SUBAPPLICATION Maehwerksklappung_DM (* Mähwerksklappung Aufgabe Febr. 2026 *)
  (* Standard: 61499-2 *)
  (* Version 1.0, 2026-02-23, Herr Lehrer *)
  PACKAGE Meins;
  IMPORT logiBUS::io::DI::logiBUS_DI::Input_I1;
  IMPORT logiBUS::io::DI::logiBUS_DI::Input_I2;
  IMPORT logiBUS::io::DI::logiBUS_DI::Input_I3;
  IMPORT logiBUS::io::DI::logiBUS_DI::Input_I4;
  IMPORT logiBUS::io::DI::logiBUS_DI::Input_I5;
  IMPORT logiBUS::io::DI::logiBUS_DI::Input_I6;
  IMPORT logiBUS::io::DI::logiBUS_DI_Events::BUTTON_PRESS_DOWN;
  IMPORT logiBUS::io::DI::logiBUS_DI_Events::BUTTON_PRESS_UP;
  IMPORT logiBUS::io::DI::logiBUS_DI_Events::BUTTON_SINGLE_CLICK;
  IMPORT logiBUS::io::DQ::logiBUS_DO::Output_Q1;
  IMPORT logiBUS::io::DQ::logiBUS_DO::Output_Q2;
  IMPORT logiBUS::io::DQ::logiBUS_DO::Output_Q3;
  IMPORT logiBUS::io::DQ::logiBUS_DO::Output_Q4;
  IMPORT logiBUS::io::DQ::logiBUS_DO::Output_Q5;
  IMPORT logiBUS::io::DQ::logiBUS_DO::Output_Q6;
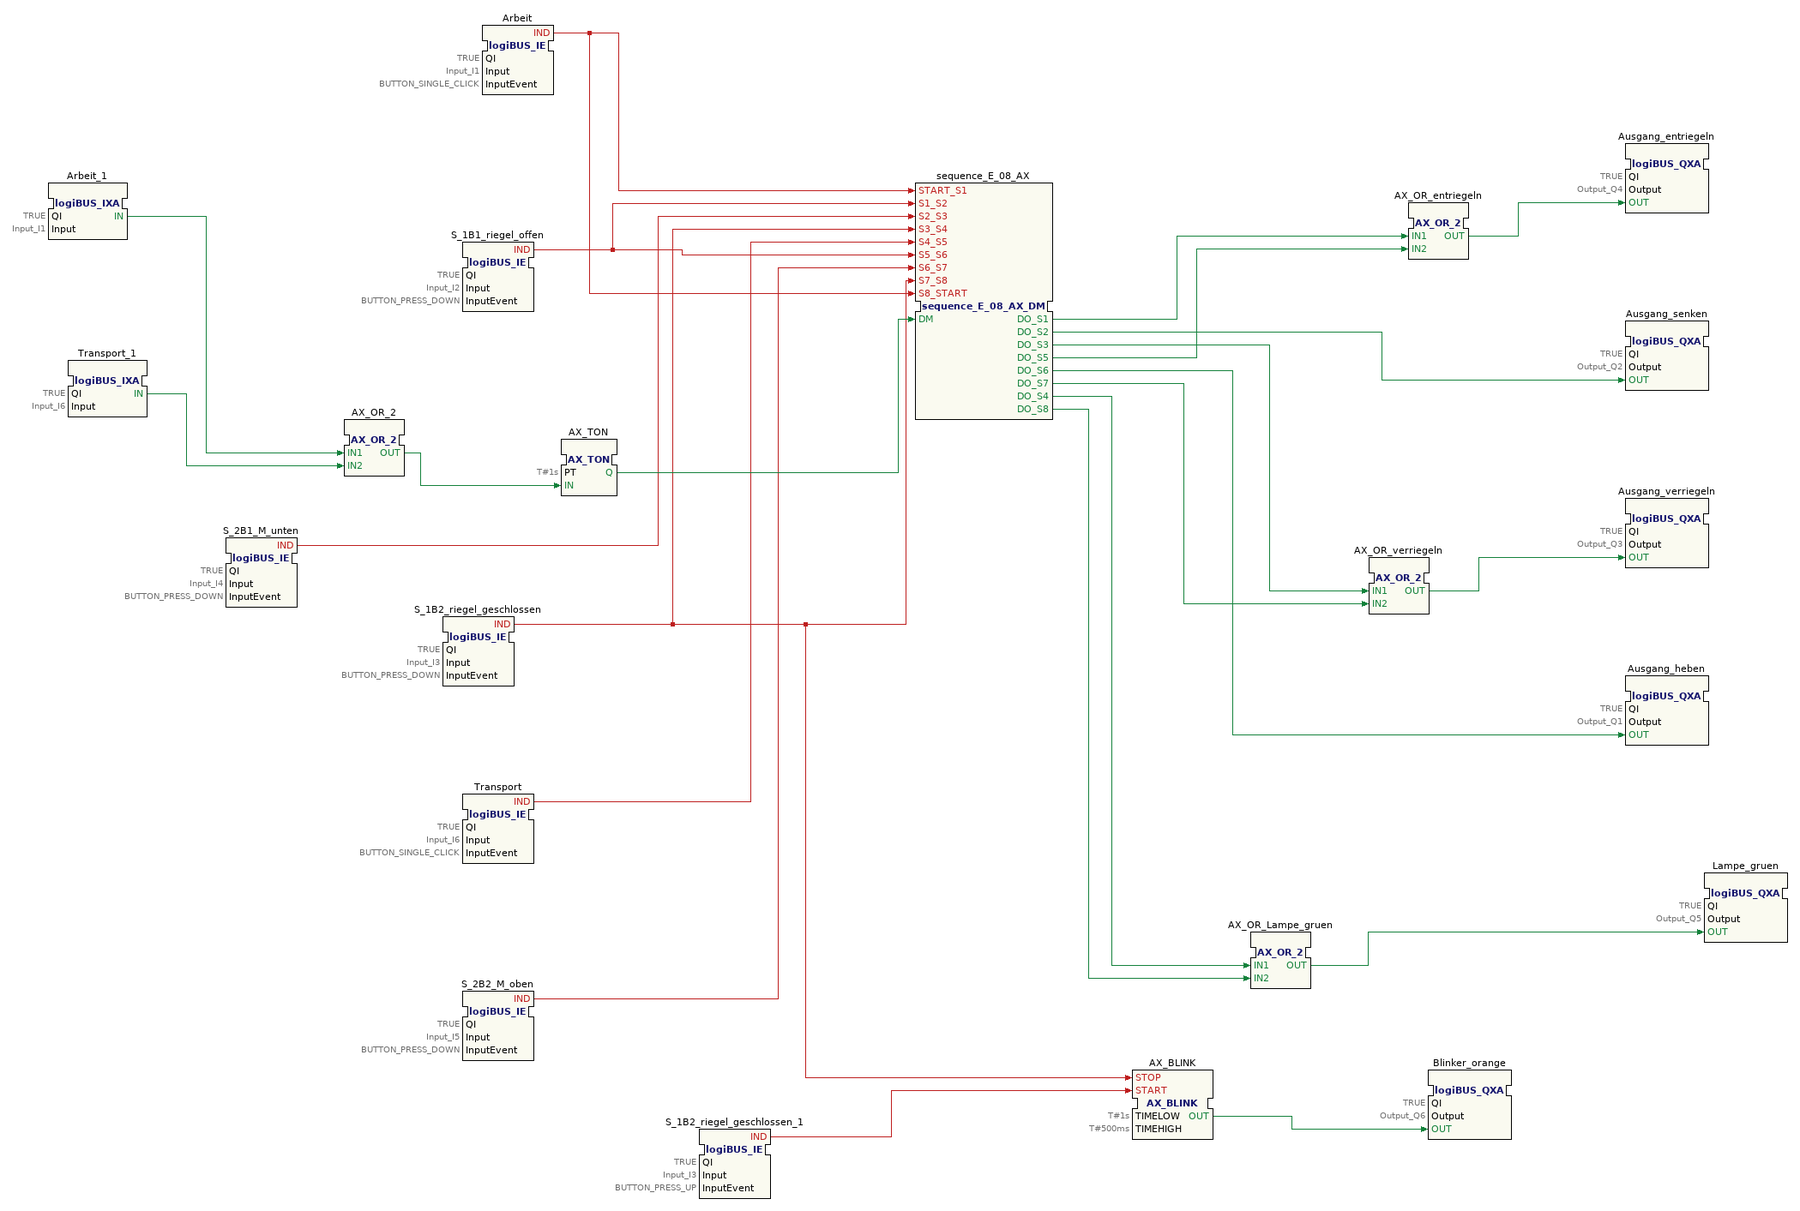
  (* UNTEN *)
  (* S4 ist der Zustand "Arbeit" *)
  (* S8 ist Zustand "Transport" *)
  FBS
    Ausgang_heben : logiBUS::io::DQ::logiBUS_QXA(QI := TRUE, Output := Output_Q1);
    Ausgang_senken : logiBUS::io::DQ::logiBUS_QXA(QI := TRUE, Output := Output_Q2);
    Ausgang_entriegeln : logiBUS::io::DQ::logiBUS_QXA(QI := TRUE, Output := Output_Q4);
    Ausgang_verriegeln : logiBUS::io::DQ::logiBUS_QXA(QI := TRUE, Output := Output_Q3);
    Lampe_gruen : logiBUS::io::DQ::logiBUS_QXA(QI := TRUE, Output := Output_Q5);
    Blinker_orange : logiBUS::io::DQ::logiBUS_QXA(QI := TRUE, Output := Output_Q6);
    Arbeit : logiBUS::io::DI::logiBUS_IE(QI := TRUE, Input := Input_I1, InputEvent := BUTTON_SINGLE_CLICK);
    S_1B1_riegel_offen : logiBUS::io::DI::logiBUS_IE(QI := TRUE, Input := Input_I2, InputEvent := BUTTON_PRESS_DOWN);
    S_1B2_riegel_geschlossen : logiBUS::io::DI::logiBUS_IE(QI := TRUE, Input := Input_I3, InputEvent := BUTTON_PRESS_DOWN);
    S_2B2_M_oben : logiBUS::io::DI::logiBUS_IE(QI := TRUE, Input := Input_I5, InputEvent := BUTTON_PRESS_DOWN);
    S_2B1_M_unten : logiBUS::io::DI::logiBUS_IE(QI := TRUE, Input := Input_I4, InputEvent := BUTTON_PRESS_DOWN);
    Transport : logiBUS::io::DI::logiBUS_IE(QI := TRUE, Input := Input_I6, InputEvent := BUTTON_SINGLE_CLICK);
    sequence_E_08_AX : logiBUS::utils::sequence::event::sequence_E_08_AX_DM;
    AX_OR_entriegeln : adapter::booleanOperators::AX_OR_2;
    AX_OR_verriegeln : adapter::booleanOperators::AX_OR_2;
    AX_OR_Lampe_gruen : adapter::booleanOperators::AX_OR_2;
    S_1B2_riegel_geschlossen_1 : logiBUS::io::DI::logiBUS_IE(QI := TRUE, Input := Input_I3, InputEvent := BUTTON_PRESS_UP);
    AX_BLINK : adapter::events::unidirectional::signals::AX_BLINK(TIMELOW := T#1s, TIMEHIGH := T#500ms);
    Arbeit_1 : logiBUS::io::DI::logiBUS_IXA(QI := TRUE, Input := Input_I1);
    Transport_1 : logiBUS::io::DI::logiBUS_IXA(QI := TRUE, Input := Input_I6);
    AX_OR_2 : adapter::booleanOperators::AX_OR_2;
    AX_TON : adapter::events::unidirectional::timers::AX_TON(PT := T#1s);
  END_FBS
  EVENT_CONNECTIONS
    Arbeit.IND TO sequence_E_08_AX.START_S1;
    S_1B1_riegel_offen.IND TO sequence_E_08_AX.S1_S2;
    S_2B1_M_unten.IND TO sequence_E_08_AX.S2_S3;
    S_1B2_riegel_geschlossen.IND TO sequence_E_08_AX.S3_S4;
    Transport.IND TO sequence_E_08_AX.S4_S5;
    S_1B1_riegel_offen.IND TO sequence_E_08_AX.S5_S6;
    S_2B2_M_oben.IND TO sequence_E_08_AX.S6_S7;
    S_1B2_riegel_geschlossen.IND TO sequence_E_08_AX.S7_S8;
    Arbeit.IND TO sequence_E_08_AX.S8_START;
    S_1B2_riegel_geschlossen.IND TO AX_BLINK.STOP;
    S_1B2_riegel_geschlossen_1.IND TO AX_BLINK.START;
  END_CONNECTIONS
  ADAPTER_CONNECTIONS
    sequence_E_08_AX.DO_S1 TO AX_OR_entriegeln.IN1;
    sequence_E_08_AX.DO_S2 TO Ausgang_senken.OUT;
    sequence_E_08_AX.DO_S3 TO AX_OR_verriegeln.IN1;
    AX_OR_entriegeln.OUT TO Ausgang_entriegeln.OUT;
    sequence_E_08_AX.DO_S5 TO AX_OR_entriegeln.IN2;
    sequence_E_08_AX.DO_S6 TO Ausgang_heben.OUT;
    AX_OR_verriegeln.OUT TO Ausgang_verriegeln.OUT;
    sequence_E_08_AX.DO_S7 TO AX_OR_verriegeln.IN2;
    AX_OR_Lampe_gruen.OUT TO Lampe_gruen.OUT;
    sequence_E_08_AX.DO_S4 TO AX_OR_Lampe_gruen.IN1;
    sequence_E_08_AX.DO_S8 TO AX_OR_Lampe_gruen.IN2;
    AX_BLINK.OUT TO Blinker_orange.OUT;
    Arbeit_1.IN TO AX_OR_2.IN1;
    Transport_1.IN TO AX_OR_2.IN2;
    AX_OR_2.OUT TO AX_TON.IN;
    AX_TON.Q TO sequence_E_08_AX.DM;
  END_CONNECTIONS
END_SUBAPPLICATION
